Fanuc KAREL source: kb00110.KL

-- PROVISIONAL review KL for V770-1; original PC SHA256 c7c4cbfead845f4dc16d9ff55850769eca782b4c32c9adac576089dde3f03359
-- Incomplete behavior may be omitted. Consult companion uncertainty JSON. Do not deploy.
PROGRAM KB00110
%NOLOCKGROUP
BEGIN
  -- UNRESOLVED_PC offsets 5-12; opcodes 9D,23
  -- UNRESOLVED_PC offsets 17-24; opcodes 9D,23
  -- UNRESOLVED_PC offsets 29-36; opcodes 9D,23
  -- UNRESOLVED_PC offsets 41-48; opcodes 9D,23
  -- UNRESOLVED_PC offsets 53-81; opcodes 27,22,22,22,22,31
  -- UNRESOLVED_PC offsets 86-90; opcodes 7F
END KB00110
